FUNCTION_BLOCK ZAppSequenceBootFault EXTENDS ZAppSequence IMPLEMENTS ZCore.ISequence
VAR
  _step : ZCore.Step(ZAppStep.BootFaultBegin, ZAppStep.BootFaultEnd);
END_VAR

IF OnStart(_step)
THEN
  // init custom sequence variables here ...
END_IF

REPEAT
  LogStep();

  CASE _step.Index OF
    (* -------------------------------------------------------------------------------------------------------------------------------- *)
    ZAppStep.BootFaultBegin:
    (* -------------------------------------------------------------------------------------------------------------------------------- *)
      _step.SetNext(ZAppStep.BootFaultEnd);
      
    (* -------------------------------------------------------------------------------------------------------------------------------- *)
    ZAppStep.BootFaultEnd:
    (* -------------------------------------------------------------------------------------------------------------------------------- *)
      SetBusy(FALSE);
      
  ELSE
    Abort('sequence contains unhandled step');
  END_CASE
UNTIL _step.IsNotRepeatable() OR_ELSE NOT Busy END_REPEAT

END_FUNCTION_BLOCK

(* stored: Version 1.1.0.1
   POU ZAppSequenceBootFault: Id {4195ac7f-36db-48a1-b509-9ee52941c536}, SpecialFunc None *)
